// TIA Portal V20 export
TYPE "UDT_Interlock_Linea_produccion"
   STRUCT
      "ENTREGA ULMA A LINEA" : Struct
         AVTF_ULMA_LINEA : Bool;
         DESC_ACT_ULMA_LINEA : Bool;
         MAN_AV_SIMUL_ULMA_LINEA : Bool;
         MAN_RET_SIMUL_ULMA_LINEA : Bool;
         PTF_LINEA_ULMA : Bool;
         FTF_LINEA_ULMA : Bool;
         MAN_AV_SIMUL_LINEA_ULMA : Bool;
         MAN_RET_SIMUL_LINEA_ULMA : Bool;
         Byte1_bit0 : Bool;
         Byte1_bit1 : Bool;
         Byte1_bit2 : Bool;
         Byte1_bit3 : Bool;
         Byte1_bit4 : Bool;
         Byte1_bit5 : Bool;
         Byte1_bit6 : Bool;
         Byte1_bit7 : Bool;
      END_STRUCT;
      "ENTREGA LINEA A ULMA" : Struct
         AVTF_LINEA_ULMA : Bool;
         DESC_ACT_LINEA_ULMA : Bool;
         MAN_AV_SIMUL_LINEA_ULMA : Bool;
         MAN_RET_SIMUL_LINEA_ULMA : Bool;
         PTF_ULMA_LINEA : Bool;
         FTF_ULMA_LINEA : Bool;
         MAN_AV_SIMUL_ULMA_LINEA : Bool;
         MAN_RET_SIMUL_ULMA_LINEA : Bool;
         Byte3_bit0 : Bool;
         Byte3_bit1 : Bool;
         Byte3_bit2 : Bool;
         Byte3_bit3 : Bool;
         Byte3_bit4 : Bool;
         Byte3_bit5 : Bool;
         Byte3_bit6 : Bool;
         Byte3_bit7 : Bool;
      END_STRUCT;
   END_STRUCT;
END_TYPE
